// TIA Portal project "w7 scl practice test miniproduction" (V15.1)

(* hardware
DEVICE "S7-1200 station_1"  S7-1200 Station
   slot 0: "Rack_0"  S7-1200 Rack  Rack  V1.0
   slot 1: "PLC_1"  CPU 1214C DC/DC/DC  6ES7 214-1AG40-0XB0  V4.1
      slot 3: "AQ 1x12BIT_1"  AQ1 signal board  6ES7 232-4HA30-0XB0  V1.0
   slot 2: "DI 8/DQ 8x24VDC_1"  6ES7 223-1BH32-0XB0  V2.0
DEVICE "HMI_1"  KTP700 Basic PN
   slot 0: "HMI_1"  KTP700 Basic PN  6AV2 123-2GB03-0AX0  15.1.0.0
   slot 1: "HMI_RT_1"  KTP700 Basic PN  6AV2 123-2GB03-0AX0  15.1.0.0
   slot 5: "HMI_1.IE_CP_1"  PROFINET Interface  15.0.1.0
      slot 1: "PROFINET Interface_1"  PROFINET Interface
         slot 1: "Port_1"  Port
DEVICE "S7-1200 station_2"  S7-1200 Station
   slot 0: "Rack_0"  S7-1200 Rack  Rack  V1.0
   slot 1: "PLC_2"  CPU 1214C DC/DC/DC  6ES7 214-1AG40-0XB0  V4.2
      slot 3: "AQ 1x12BIT_1"  AQ1 signal board  6ES7 232-4HA30-0XB0  V1.0
   slot 2: "DI 8/DQ 8x24VDC_1"  6ES7 223-1BH32-0XB0  V2.0
DEVICE "S7-1200 station_3"  S7-1200 Station
   slot 0: "Rack_0"  S7-1200 Rack  Rack  V1.0
   slot 1: "PLC_3"  CPU 1214C DC/DC/DC  6ES7 214-1AG40-0XB0  V4.1
      slot 3: "AQ 1x12BIT_1"  AQ1 signal board  6ES7 232-4HA30-0XB0  V1.0
   slot 2: "DI 8/DQ 8x24VDC_1"  6ES7 223-1BH32-0XB0  V2.0
*)

// ===== PLC "PLC_1"  CPU 1214C DC/DC/DC =====

VAR_GLOBAL   // PLC tag table "Default tag table"
   "SA2" AT %I0.1 : Bool;
   "SA1" AT %I0.2 : Bool;
   "vacuum built" AT %I0.3 : Bool;
   "SB2" AT %I0.4 : Bool;
   "SB1" AT %I0.5 : Bool;
   "no workpiece" AT %I0.6 : Bool;
   "A+" AT %Q0.0 : Bool;
   "turn on vacuum" AT %Q0.1 : Bool;
   "turn on air" AT %Q0.2 : Bool;
   "B+" AT %Q0.3 : Bool;
   "B-" AT %Q0.4 : Bool;
   "green" AT %Q0.5 : Bool;
   "yellow" AT %Q0.6 : Bool;
   "red" AT %Q0.7 : Bool;
   "station 2 ready" AT %I0.7 : Bool;
END_VAR

DATA_BLOCK "Block_1_DB"   // DB1
{ S7_Optimized_Access := 'TRUE' }
VERSION : 0.1
// stored: InstanceOfName Block_1
"Block_1"
BEGIN
END_DATA_BLOCK

FUNCTION_BLOCK "Block_1"   // FB1, SCL
{ S7_Optimized_Access := 'TRUE' }
VERSION : 0.1
   VAR
      my_steps : Int;
      "timer" : TON_TIME;
   END_VAR
BEGIN
   CASE #my_steps OF
       0:
           RESET_TIMER(#timer);
           "A+" := False;   //reset all 
           "B+" := False;
           "B-" := True;
           "green" := FALSE;
           "yellow" := TRUE;
           "turn on vacuum" := False;
           "turn on air" := False;
           IF NOT "no workpiece" AND "SA2" AND "SB1" THEN //wait until there is a product
               "green" := TRUE;
               "yellow" := FALSE;
               #my_steps := #my_steps + 1;                   
               ;                                
           END_IF;
           ;
       1:
           "A+" := True;   //extend A cylinder to push out product
               IF "SA1" THEN       //if cylinder pushed out product move on
                   #my_steps := #my_steps + 1;
               END_IF;
               ;
       2:
           "B-" := FALSE;  //come TO pick up product
           "B+" := True;
           IF "SB2" THEN  //when arrived move on
               #my_steps := #my_steps + 1; 
           END_IF;

       3:
           IF "station 2 ready" THEN        //when next station not busy anymore
               #my_steps := #my_steps + 1;
               ;
           END_IF;

       4:
           "turn on vacuum" := True;   //turn vacuum on
           IF "vacuum built" THEN      //when vacuum built up 
               #my_steps := #my_steps + 1;    //move on
               ;
           END_IF;
           ;


       5: 
           "A+" := FALSE; //retract A cylinder
           IF "SA2" THEN
               "B+" := False;      //Assuming product picked move it downstream
               "B-" := True;
               IF "SB1" THEN
                   #my_steps := #my_steps + 1;
                   ;
               END_IF;
               ;
           END_IF;

       6:
           "turn on vacuum" := False; //when product arrived drop it
           "turn on air" := True;
           IF NOT "vacuum built" THEN
                   #my_steps := #my_steps + 1;
                   ;

               END_IF;

       7:

           "B+" := True;      //Assuming product picked move it downstream
           "B-" := False;
           "turn on air" := 0;
           IF "SB2" THEN
               #my_steps := 0;
               ;
           END_IF;            ;
       ELSE  // Statement section ELSE
           ;
   END_CASE;
END_FUNCTION_BLOCK

ORGANIZATION_BLOCK "Main"   // OB1, LAD, ProgramCycle
TITLE = "Main Program Sweep (Cycle)"
{ S7_Optimized_Access := 'TRUE' }
VERSION : 0.1
   VAR_INPUT
      Initial_Call : Bool;   // Initial call of this OB
      Remanence : Bool;   // =True, if remanent data are available
   END_VAR
BEGIN

REGION Network 1
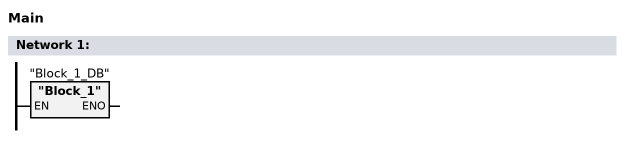
   RUNG wire#powerrail
      "Block_1_DB"()
   END_RUNG
   // the same network as SCL:
   "Block_1_DB"();   // "Block_1"
END_REGION
END_ORGANIZATION_BLOCK

// ===== PLC "PLC_2"  CPU 1214C DC/DC/DC =====

VAR_GLOBAL   // PLC tag table "Default tag table"
   "product at processing point" AT %I0.0 : Bool;
   "product not at end" AT %I0.1 : Bool;
   "horizontal retracted" AT %I0.2 : Bool;
   "vertical extended" AT %I0.3 : Bool;
   "vacuum biult" AT %I0.4 : Bool;
   "horizontal extended" AT %I0.5 : Bool;
   "product arrived" AT %I0.6 : Bool;
   "station3ready" AT %I0.7 : Bool;
   "conveyor ON" AT %Q0.0 : Bool;
   "Horizontal -" AT %Q0.1 : Bool;
   "Horizontal +" AT %Q0.2 : Bool;
   "Vertical +" AT %Q0.3 : Bool;
   "turn on vacuum" AT %Q0.4 : Bool;
   "stopper on" AT %Q0.5 : Bool;
   "station 2 is busy" AT %Q0.6 : Bool;
END_VAR

DATA_BLOCK "Block_1_DB"   // DB1
{ S7_Optimized_Access := 'TRUE' }
VERSION : 0.1
// stored: InstanceOfName Block_1
"Block_1"
BEGIN
END_DATA_BLOCK

DATA_BLOCK "Block_1_DB_1"   // DB2
{ S7_Optimized_Access := 'TRUE' }
VERSION : 0.1
// stored: InstanceOfName Block_1
"Block_1"
BEGIN
END_DATA_BLOCK

DATA_BLOCK "Block_1_DB_2"   // DB3
{ S7_Optimized_Access := 'TRUE' }
VERSION : 0.1
// stored: InstanceOfName Block_1
"Block_1"
BEGIN
END_DATA_BLOCK

FUNCTION_BLOCK "Block_1"   // FB1, SCL
{ S7_Optimized_Access := 'TRUE' }
VERSION : 0.1
   VAR
      my_steps2 : Int;
      "timer" : TON_TIME;
   END_VAR
BEGIN
   CASE #my_steps2 OF
       0:
           "conveyor ON" := FALSE;     //reset all
           "Vertical +" := FALSE;
           "Horizontal -" := TRUE;
           "Horizontal +" := FALSE;
           "turn on vacuum" := FALSE;
           "stopper on" := FALSE;
           "station 2 is busy" := FALSE;
           IF "product arrived" THEN       //when product arrives move to next step

               #my_steps2 := #my_steps2 + 1;
               ;
           END_IF;

           ;
       1:
           "conveyor ON" := TRUE;      //turn on conveyor and stopper
           "stopper on" := TRUE;
           "station 2 is busy" := TRUE;
           IF "product at processing point" THEN      //when arrived to processing point move on
               #my_steps2 := #my_steps2 + 1;
               ;
           END_IF;

       2:
           #timer(IN := 1,     //wait for a second so product gets in position
                  PT := T#1s);
           IF #timer.Q THEN
               RESET_TIMER(#timer);
               "conveyor ON" := FALSE;     //conveyor off
               #my_steps2 := #my_steps2 + 1;
               ;
           END_IF;

       3:
           IF "horizontal retracted" AND NOT "vertical extended" THEN //when cylinders in right position
               "Vertical +" := TRUE; //vertical cylindr down
               #my_steps2 := #my_steps2 + 1;
               ;
           END_IF;

       4:
           IF "vertical extended" THEN //when cylinder in position
               "turn on vacuum" := TRUE;        //vacuum
               #my_steps2 := #my_steps2 + 1;
               ;
           END_IF;
       5:
           IF "vacuum biult" THEN      //if vacuum built
               "Vertical +" := FALSE;  //pick up lid
               #my_steps2 := #my_steps2 + 1;
               ;
           END_IF;

       6:
           IF NOT "vertical extended" THEN     //when vertical is up
               "Horizontal +" := TRUE;         //horizontal extract
               "Horizontal -" := FALSE;
               #my_steps2 := #my_steps2 + 1;
               ;
           END_IF;

       7:
           IF "horizontal extended" THEN      //when product over the conveyor
               "Vertical +" := TRUE;        //put down product
               #my_steps2 := #my_steps2 + 1;
               ;
           END_IF;

       8:
           IF "vertical extended" THEN     //when lid placed on
               "turn on vacuum" := FALSE;      // turn vacuum off
               #my_steps2 := #my_steps2 + 1;
               ;
           END_IF;
       9:
           IF NOT "vacuum biult" THEN
               "Vertical +" := FALSE;
               #my_steps2 := #my_steps2 + 1;
               ;
           END_IF;
       10:
           IF NOT "vertical extended" THEN
               "Horizontal +" := FALSE;
               "Horizontal -" := TRUE;
               #my_steps2 := #my_steps2 + 1;
               ;
           END_IF;

       11:
           IF "station3ready" THEN
               #my_steps2 := #my_steps2 + 1;
               ;
           END_IF;


       12:
           IF NOT "vertical extended" AND "horizontal retracted" THEN      //when cylinders both retracted
               "stopper on" := FALSE;                                       //turn stopper to let product go
               #my_steps2 := #my_steps2 + 1;
               ;
           END_IF;

       13:
           IF NOT "stopper on" THEN
               "conveyor ON" := TRUE;
               #my_steps2 := #my_steps2 + 1;
               ;
           END_IF;
       14:
           IF NOT "product not at end" THEN        //when product at end of conveyor wait a bit
               #timer(IN := 1,
                      PT := T#1s);
               #my_steps2 := #my_steps2 + 1;
           END_IF;
           ;
       15:        
           IF #timer.Q THEN
                   RESET_TIMER(#timer);
                   #my_steps2 := 0;        //all done, go back reset everything to initial position  
                   ;                      //and tell station1 thet station 2 not busy anymore

           END_IF;

       ELSE  // Statement section ELSE
           ;
   END_CASE;
END_FUNCTION_BLOCK

ORGANIZATION_BLOCK "Main"   // OB1, LAD, ProgramCycle
TITLE = "Main Program Sweep (Cycle)"
{ S7_Optimized_Access := 'TRUE' }
VERSION : 0.1
   VAR_INPUT
      Initial_Call : Bool;   // Initial call of this OB
      Remanence : Bool;   // =True, if remanent data are available
   END_VAR
BEGIN

REGION Network 1
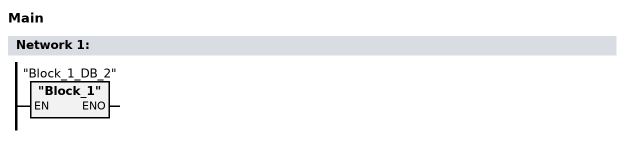
   RUNG wire#powerrail
      "Block_1_DB_2"()
   END_RUNG
   // the same network as SCL:
   "Block_1_DB_2"();   // "Block_1"
END_REGION
END_ORGANIZATION_BLOCK

// ===== PLC "PLC_3"  CPU 1214C DC/DC/DC =====

VAR_GLOBAL   // PLC tag table "Default tag table"
   "work piece available" AT %I0.0 : Bool;
   "metal sensor" AT %I0.1 : Bool;
   "not black" AT %I0.2 : Bool;
   "product slided down" AT %I0.3 : Bool;
   "A extended" AT %I0.4 : Bool;
   "A retracted" AT %I0.5 : Bool;
   "B extended" AT %I0.6 : Bool;
   "B retracted" AT %I0.7 : Bool;
   "turn on conveyor" AT %Q0.0 : Bool;
   "extend A" AT %Q0.1 : Bool;
   "extend B" AT %Q0.2 : Bool;
   "retract stopper" AT %Q0.3 : Bool;
   "green" AT %Q0.4 : Bool;
   "yellow" AT %Q0.5 : Bool;
   "red" AT %Q0.6 : Bool;
   "station 3 busy" AT %Q0.7 : Bool;
END_VAR

DATA_BLOCK "Block_1_DB"   // DB1
{ S7_Optimized_Access := 'TRUE' }
VERSION : 0.1
// stored: InstanceOfName Block_1
"Block_1"
BEGIN
END_DATA_BLOCK

FUNCTION_BLOCK "Block_1"   // FB1, SCL
{ S7_Optimized_Access := 'TRUE' }
VERSION : 0.1
   VAR
      my_steps2 : Int;
      "timer" : TON_TIME;
   END_VAR
BEGIN
   CASE #my_steps2 OF
       0:
           "turn on conveyor" := FALSE;        //reset everything
           "extend A" := FALSE;
           "extend B" := FALSE;
           "retract stopper" := FALSE;
           "station 3 busy" := FALSE;
           "green" := FALSE;
           "red" := FALSE;
           "yellow" := TRUE;
           IF "work piece available" THEN      //when there is product start conveyor
               "station 3 busy" := TRUE;
               "green" := TRUE;
               "red" := FALSE;
               "yellow" := FALSE;
               "turn on conveyor" := TRUE;
               #my_steps2 := 5;
               ;
           END_IF;
           ;

       5:
           IF "A retracted" AND "B retracted" THEN //when cylinders both retracted move on
               #my_steps2 := 10;
               ;
           END_IF;
           ;
       10:
           #timer(IN := 1,     //wait for a second so product gets in position
                  PT := T#2s);
           IF #timer.Q THEN
               RESET_TIMER(#timer);
               #my_steps2 := 20;
               ;
           END_IF;
           ;
       20:    
           IF "not black" AND NOT "metal sensor" THEN      //if not black and not metal (RED)
               "extend B" := TRUE;                         //extend A cyliner
               #my_steps2 := 30;
               ;
           END_IF;

           IF "not black" AND "metal sensor" THEN      //if not black and metal (SYLVER)
               "extend A" := TRUE;                     //extend cylinder 2
               #my_steps2 := 40;
               ;
           END_IF;

           IF NOT "not black" AND NOT "metal sensor" THEN      //if  black and not metal (BLack)
               "retract stopper" := TRUE;                      //let product go
               #my_steps2 := 100;
               ;
           END_IF;
           ;
       30:
           IF "B extended" THEN                                //if cylinder 2 extended position
               "retract stopper" := True;                      //let it go forward
               #my_steps2 := 100;
               ;
           END_IF;
           ;
       40:
           IF "A extended" THEN                                //if extended
               "retract stopper" := True;                      //let it go forward
               #my_steps2 := 100;
               ;
           END_IF;
           ;
       100:
           IF "product slided down" THEN       //when left slide reset all and wait for more products
               #my_steps2 := 0;
               ;
           END_IF;
           ;
       ELSE  // Statement section ELSE
           ;
   END_CASE;
END_FUNCTION_BLOCK

ORGANIZATION_BLOCK "Main"   // OB1, LAD, ProgramCycle
TITLE = "Main Program Sweep (Cycle)"
{ S7_Optimized_Access := 'TRUE' }
VERSION : 0.1
   VAR_INPUT
      Initial_Call : Bool;   // Initial call of this OB
      Remanence : Bool;   // =True, if remanent data are available
   END_VAR
BEGIN

REGION Network 1
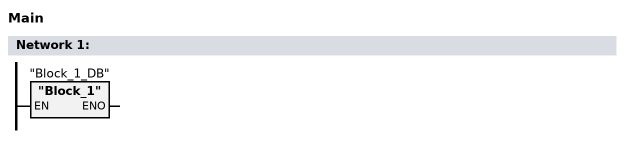
   RUNG wire#powerrail
      "Block_1_DB"()
   END_RUNG
   // the same network as SCL:
   "Block_1_DB"();   // "Block_1"
END_REGION
END_ORGANIZATION_BLOCK

(* ===== HMI "HMI_RT_1" =====
system functions are stored by id; their names below are inferred from use

HMI tags "Default tag table"
   "Tag_ScreenNumber" : UInt, internal
   "am/pm_DB_time" : DateTime, internal

Template "Template_1" 800x480
   Button "Exit" at 714,429 size 71x50; TextOff 'Exit'; PictureOff "ExitRuntime_KTP700_Basic_PN_TR"; PictureOn "ExitRuntime_KTP700_Basic_PN_TR"
      on Release: StopRuntime(0)
   Button "Template_Button" at 614,429 size 71x50; TextOff 'Text'
   Button "Template_Button_1" at 514,429 size 71x50; TextOff 'Text'
   Button "Template_Button_2" at 414,429 size 71x50; TextOff 'Text'
   Button "Template_Button_3" at 314,429 size 71x50; TextOff 'Text'
   Button "Template_Button_4" at 214,429 size 71x50; TextOff 'Text'
   Button "Template_Button_5" at 114,429 size 71x50; TextOff 'Text'
   Button "Start screen" at 14,429 size 71x50; TextOff 'Start screen'; PictureOff "NavigateHome_KTP700_Basic_PN_TR"; PictureOn "NavigateHome_KTP700_Basic_PN_TR"
      on Release: ActivateScreen("Root screen", 0)
   SymbolicIOField "Symbolic_IO_Field_Screen" at 93,9 size 600x33; TextOff '0'; TextOn '1'; TextList "TextList_ScreenNames"
      ProcessValue <- "Tag_ScreenNumber"
      on Change: ActivateScreenByNumber("Tag_ScreenNumber", 0)
   DateTimeField "HmiScreenItemData" at 695,25 size 105x25
   DateTimeField "HmiScreenItemData_1" at 695,0 size 105x25
   GraphicView "Logo" at 0,0 size 91x51; Picture "Logo of HMI_1"

screen "Root screen" 800x480, template "Template_1"
   on GenerateScreen: SetTag("Tag_ScreenNumber", 1)
   TextField "HmiScreenItemData" at 80,225 size 640x25; Text 'Welcome to HMI_1 (KTP700 Basic+ PN)!'
*)